(* PLC project PhysicsSimulator, Nammo OpenPLC 1 *)
(* stored: creationDateTime 2026-02-21T00:00:00, modificationDateTime 2026-02-21T00:00:00 *)

TYPE STATION_T : STRUCT
  number : INT;
  x_mm : REAL;
  station_type : INT;
  device_delay_s : REAL;
  dropping_time_s : REAL;
END_STRUCT;
END_TYPE

TYPE PHYSICS_2D_T : STRUCT
  x_accel_s : REAL;
  x_decel_s : REAL;
  x_max_mm_s : REAL;
  z_total_mm : REAL;
  z_slow_dry_mm : REAL;
  z_slow_wet_mm : REAL;
  z_slow_end_mm : REAL;
  z_slow_mm_s : REAL;
  z_fast_mm_s : REAL;
  drip_delay_s : REAL;
  avoid_mm : REAL;
END_STRUCT;
END_TYPE

TYPE TRANSPORTER_CFG_T : STRUCT
  id : INT;
  start_station : INT;
  x_min_limit : REAL;
  x_max_limit : REAL;
  phys2d : PHYSICS_2D_T;
END_STRUCT;
END_TYPE

TYPE TRANSPORTER_STATE_T : STRUCT
  active : BOOL;
  phase : INT;
  z_stage : INT;
  x_mm : REAL;
  z_mm : REAL;
  vel_x : REAL;
  vel_z : REAL;
  current_station : INT;
  lift_station_target : INT;
  sink_station_target : INT;
  target_x : REAL;
  x_min_limit : REAL;
  x_max_limit : REAL;
  z_timer_s : REAL;
END_STRUCT;
END_TYPE

FUNCTION IsWetStationType : BOOL
  VAR_INPUT
    station_type : INT;
  END_VAR

            IsWetStationType := (station_type = 1) OR (station_type = 11);
          
END_FUNCTION

FUNCTION_BLOCK FB_StationLookup
  VAR_INPUT
    station_number : INT;
  END_VAR
  VAR_OUTPUT
    found : BOOL;
    idx : INT;
    x_mm : REAL;
    stype : INT;
    device_delay_s : REAL;
    dropping_time_s : REAL;
  END_VAR
  VAR_EXTERNAL
    g_station_count : INT;
    g_stations : ARRAY[1..21] OF STATION_T;
  END_VAR
  VAR
    i : INT;
    tmp_st : STATION_T;
  END_VAR

            found := FALSE;
idx := 0;
x_mm := 0.0;
stype := 0;
device_delay_s := 0.0;
dropping_time_s := 0.0;

FOR i := 1 TO g_station_count DO
  tmp_st := g_stations[i];
  IF tmp_st.number = station_number THEN
    found := TRUE;
    idx := i;
    x_mm := tmp_st.x_mm;
    stype := tmp_st.station_type;
    device_delay_s := tmp_st.device_delay_s;
    dropping_time_s := tmp_st.dropping_time_s;
    RETURN;
  END_IF;
END_FOR;
          
END_FUNCTION_BLOCK

FUNCTION_BLOCK FB_XMotion
  VAR_INPUT
    delta_t : REAL;
    x_target : REAL;
    x_min : REAL;
    x_max : REAL;
    v_max : REAL;
    t_acc : REAL;
    t_dec : REAL;
  END_VAR
  VAR_IN_OUT
    x_pos : REAL;
    v_x : REAL;
  END_VAR
  VAR_OUTPUT
    arrived : BOOL;
  END_VAR
  VAR
    drive_target : REAL;
    distance : REAL;
    dir : REAL;
    a_acc : REAL;
    a_dec : REAL;
    brake_dist : REAL;
    new_vel : REAL;
    travel : REAL;
  END_VAR

            IF (x_max > x_min) THEN
  IF x_pos < x_min THEN
    drive_target := x_min;
  ELSIF x_pos > x_max THEN
    drive_target := x_max;
  ELSE
    IF x_target < x_min THEN
      drive_target := x_min;
    ELSIF x_target > x_max THEN
      drive_target := x_max;
    ELSE
      drive_target := x_target;
    END_IF;
  END_IF;
ELSE
  drive_target := x_target;
END_IF;

arrived := ABS(x_pos - drive_target) <= 3.0;
IF arrived THEN
  x_pos := drive_target;
  v_x := 0.0;
  RETURN;
END_IF;

IF t_acc <= 0.0 THEN t_acc := 0.001; END_IF;
IF t_dec <= 0.0 THEN t_dec := 0.001; END_IF;
IF v_max < 0.0 THEN v_max := 0.0; END_IF;

a_acc := v_max / t_acc;
a_dec := v_max / t_dec;

dir := 1.0;
IF drive_target < x_pos THEN
  dir := -1.0;
END_IF;

distance := ABS(drive_target - x_pos);

IF a_dec > 0.0 THEN
  brake_dist := (v_x * v_x) / (2.0 * a_dec);
ELSE
  brake_dist := 0.0;
END_IF;

IF brake_dist >= distance THEN
  new_vel := v_x - a_dec * delta_t;
  IF new_vel < 0.0 THEN new_vel := 0.0; END_IF;
ELSE
  new_vel := v_x + a_acc * delta_t;
  IF new_vel > v_max THEN new_vel := v_max; END_IF;
END_IF;

travel := new_vel * delta_t;
IF travel >= distance THEN
  x_pos := drive_target;
  v_x := 0.0;
  arrived := TRUE;
ELSE
  x_pos := x_pos + dir * travel;
  v_x := new_vel;
  arrived := FALSE;
END_IF;
          
END_FUNCTION_BLOCK

PROGRAM PLC_PRG
  VAR_EXTERNAL
    g_station_count : INT;
    g_stations : ARRAY[1..21] OF STATION_T;
    g_cfg : ARRAY[1..10] OF TRANSPORTER_CFG_T;
    g_state : ARRAY[1..10] OF TRANSPORTER_STATE_T;
    g_cmd_start : ARRAY[1..10] OF BOOL;
    g_cmd_lift_station : ARRAY[1..10] OF INT;
    g_cmd_sink_station : ARRAY[1..10] OF INT;
  END_VAR
  VAR
    init_done : BOOL := FALSE;
    i : INT;
    idx : INT;
    station_type : INT;
    device_delay : REAL;
    drop_time : REAL;
    slow_start : REAL;
    arrived_x : BOOL;
    nearest_num : INT;
    min_dist : REAL;
    dx : REAL;
    tmp_x : REAL;
    tmp_vx : REAL;
    fb_x1 : FB_XMotion;
    fb_x2 : FB_XMotion;
    lookup : FB_StationLookup;
  END_VAR

            IF NOT init_done THEN
  g_station_count := 21;

  g_stations[1].number := 101;
  g_stations[1].x_mm := 100.0;
  g_stations[1].station_type := 22;
  g_stations[1].device_delay_s := 0.0;
  g_stations[1].dropping_time_s := 0.0;

  g_stations[2].number := 102;
  g_stations[2].x_mm := 1550.0;
  g_stations[2].station_type := 30;
  g_stations[2].device_delay_s := 0.0;
  g_stations[2].dropping_time_s := 0.0;

  g_stations[3].number := 103;
  g_stations[3].x_mm := 3000.0;
  g_stations[3].station_type := 30;
  g_stations[3].device_delay_s := 0.0;
  g_stations[3].dropping_time_s := 0.0;

  g_stations[4].number := 104;
  g_stations[4].x_mm := 4450.0;
  g_stations[4].station_type := 0;
  g_stations[4].device_delay_s := 3.0;
  g_stations[4].dropping_time_s := 0.0;

  g_stations[5].number := 105;
  g_stations[5].x_mm := 5900.0;
  g_stations[5].station_type := 0;
  g_stations[5].device_delay_s := 3.0;
  g_stations[5].dropping_time_s := 0.0;

  g_stations[6].number := 106;
  g_stations[6].x_mm := 7350.0;
  g_stations[6].station_type := 0;
  g_stations[6].device_delay_s := 3.0;
  g_stations[6].dropping_time_s := 0.0;

  g_stations[7].number := 107;
  g_stations[7].x_mm := 8800.0;
  g_stations[7].station_type := 1;
  g_stations[7].device_delay_s := 3.0;
  g_stations[7].dropping_time_s := 10.0;

  g_stations[8].number := 108;
  g_stations[8].x_mm := 10250.0;
  g_stations[8].station_type := 1;
  g_stations[8].device_delay_s := 0.0;
  g_stations[8].dropping_time_s := 10.0;

  g_stations[9].number := 109;
  g_stations[9].x_mm := 11700.0;
  g_stations[9].station_type := 1;
  g_stations[9].device_delay_s := 0.0;
  g_stations[9].dropping_time_s := 10.0;

  g_stations[10].number := 110;
  g_stations[10].x_mm := 13150.0;
  g_stations[10].station_type := 1;
  g_stations[10].device_delay_s := 0.0;
  g_stations[10].dropping_time_s := 10.0;

  g_stations[11].number := 111;
  g_stations[11].x_mm := 14600.0;
  g_stations[11].station_type := 1;
  g_stations[11].device_delay_s := 0.0;
  g_stations[11].dropping_time_s := 10.0;

  g_stations[12].number := 112;
  g_stations[12].x_mm := 16050.0;
  g_stations[12].station_type := 1;
  g_stations[12].device_delay_s := 3.0;
  g_stations[12].dropping_time_s := 10.0;

  g_stations[13].number := 113;
  g_stations[13].x_mm := 17500.0;
  g_stations[13].station_type := 1;
  g_stations[13].device_delay_s := 0.0;
  g_stations[13].dropping_time_s := 10.0;

  g_stations[14].number := 114;
  g_stations[14].x_mm := 18950.0;
  g_stations[14].station_type := 32;
  g_stations[14].device_delay_s := 0.0;
  g_stations[14].dropping_time_s := 0.0;

  g_stations[15].number := 115;
  g_stations[15].x_mm := 20400.0;
  g_stations[15].station_type := 0;
  g_stations[15].device_delay_s := 3.0;
  g_stations[15].dropping_time_s := 10.0;

  g_stations[16].number := 116;
  g_stations[16].x_mm := 21850.0;
  g_stations[16].station_type := 1;
  g_stations[16].device_delay_s := 3.0;
  g_stations[16].dropping_time_s := 10.0;

  g_stations[17].number := 117;
  g_stations[17].x_mm := 23300.0;
  g_stations[17].station_type := 1;
  g_stations[17].device_delay_s := 0.0;
  g_stations[17].dropping_time_s := 10.0;

  g_stations[18].number := 118;
  g_stations[18].x_mm := 24750.0;
  g_stations[18].station_type := 1;
  g_stations[18].device_delay_s := 0.0;
  g_stations[18].dropping_time_s := 10.0;

  g_stations[19].number := 119;
  g_stations[19].x_mm := 26200.0;
  g_stations[19].station_type := 30;
  g_stations[19].device_delay_s := 0.0;
  g_stations[19].dropping_time_s := 0.0;

  g_stations[20].number := 120;
  g_stations[20].x_mm := 27650.0;
  g_stations[20].station_type := 30;
  g_stations[20].device_delay_s := 0.0;
  g_stations[20].dropping_time_s := 0.0;

  g_stations[21].number := 121;
  g_stations[21].x_mm := 29100.0;
  g_stations[21].station_type := 1;
  g_stations[21].device_delay_s := 0.0;
  g_stations[21].dropping_time_s := 10.0;

  g_cfg[1].id := 1;
  g_cfg[1].start_station := 101;
  g_cfg[1].x_min_limit := 100.0;
  g_cfg[1].x_max_limit := 20600.0;
  g_cfg[1].phys2d.x_accel_s := 1.5;
  g_cfg[1].phys2d.x_decel_s := 1.5;
  g_cfg[1].phys2d.x_max_mm_s := 500.0;
  g_cfg[1].phys2d.z_total_mm := 2500.0;
  g_cfg[1].phys2d.z_slow_dry_mm := 300.0;
  g_cfg[1].phys2d.z_slow_wet_mm := 1000.0;
  g_cfg[1].phys2d.z_slow_end_mm := 50.0;
  g_cfg[1].phys2d.z_slow_mm_s := 100.0;
  g_cfg[1].phys2d.z_fast_mm_s := 200.0;
  g_cfg[1].phys2d.drip_delay_s := 5.0;
  g_cfg[1].phys2d.avoid_mm := 2000.0;

  g_cfg[2].id := 2;
  g_cfg[2].start_station := 118;
  g_cfg[2].x_min_limit := 14300.0;
  g_cfg[2].x_max_limit := 29100.0;
  g_cfg[2].phys2d.x_accel_s := 1.5;
  g_cfg[2].phys2d.x_decel_s := 1.5;
  g_cfg[2].phys2d.x_max_mm_s := 500.0;
  g_cfg[2].phys2d.z_total_mm := 2500.0;
  g_cfg[2].phys2d.z_slow_dry_mm := 300.0;
  g_cfg[2].phys2d.z_slow_wet_mm := 1000.0;
  g_cfg[2].phys2d.z_slow_end_mm := 50.0;
  g_cfg[2].phys2d.z_slow_mm_s := 100.0;
  g_cfg[2].phys2d.z_fast_mm_s := 200.0;
  g_cfg[2].phys2d.drip_delay_s := 5.0;
  g_cfg[2].phys2d.avoid_mm := 2000.0;

  FOR i := 1 TO 10 DO
    IF i <= 2 THEN
      g_state[i].active := TRUE;
    ELSE
      g_state[i].active := FALSE;
    END_IF;
    g_state[i].phase := 0;
    g_state[i].z_stage := 0;
    g_state[i].vel_x := 0.0;
    g_state[i].vel_z := 0.0;
    g_state[i].z_timer_s := 0.0;
    g_state[i].x_min_limit := g_cfg[i].x_min_limit;
    g_state[i].x_max_limit := g_cfg[i].x_max_limit;

    lookup(station_number := g_cfg[i].start_station);
    IF lookup.found THEN
      g_state[i].x_mm := lookup.x_mm;
      g_state[i].current_station := g_cfg[i].start_station;
    ELSE
      g_state[i].x_mm := 0.0;
      g_state[i].current_station := 0;
    END_IF;
    g_state[i].z_mm := 0.0;
  END_FOR;

  init_done := TRUE;
END_IF;

FOR i := 1 TO 10 DO
  IF g_state[i].active THEN

  IF (g_state[i].phase = 0) AND g_cmd_start[i] THEN
    g_state[i].lift_station_target := g_cmd_lift_station[i];
    g_state[i].sink_station_target := g_cmd_sink_station[i];
    lookup(station_number := g_state[i].lift_station_target);
    g_state[i].target_x := lookup.x_mm;
    g_state[i].phase := 1;
    g_state[i].z_stage := 0;
    g_state[i].z_timer_s := 0.0;
  END_IF;

  IF g_state[i].phase = 1 THEN
    tmp_x := g_state[i].x_mm;
    tmp_vx := g_state[i].vel_x;
    IF i = 1 THEN
      fb_x1(
        delta_t := 0.02,
        x_target := g_state[i].target_x,
        x_min := g_state[i].x_min_limit,
        x_max := g_state[i].x_max_limit,
        v_max := g_cfg[i].phys2d.x_max_mm_s,
        t_acc := g_cfg[i].phys2d.x_accel_s,
        t_dec := g_cfg[i].phys2d.x_decel_s,
        x_pos := tmp_x,
        v_x := tmp_vx
      );
      arrived_x := fb_x1.arrived;
    ELSIF i = 2 THEN
      fb_x2(
        delta_t := 0.02,
        x_target := g_state[i].target_x,
        x_min := g_state[i].x_min_limit,
        x_max := g_state[i].x_max_limit,
        v_max := g_cfg[i].phys2d.x_max_mm_s,
        t_acc := g_cfg[i].phys2d.x_accel_s,
        t_dec := g_cfg[i].phys2d.x_decel_s,
        x_pos := tmp_x,
        v_x := tmp_vx
      );
      arrived_x := fb_x2.arrived;
    END_IF;
    g_state[i].x_mm := tmp_x;
    g_state[i].vel_x := tmp_vx;

    IF arrived_x THEN
      g_state[i].current_station := g_state[i].lift_station_target;
      lookup(station_number := g_state[i].lift_station_target);
      device_delay := lookup.device_delay_s;
      drop_time := lookup.dropping_time_s;
      g_state[i].z_timer_s := device_delay + drop_time;
      g_state[i].z_stage := 1;
      g_state[i].phase := 2;
    END_IF;
  END_IF;

  IF g_state[i].phase = 2 THEN
    lookup(station_number := g_state[i].lift_station_target);
    station_type := lookup.stype;
    IF IsWetStationType(station_type) THEN
      slow_start := g_cfg[i].phys2d.z_slow_wet_mm;
    ELSE
      slow_start := g_cfg[i].phys2d.z_slow_dry_mm;
    END_IF;

    CASE g_state[i].z_stage OF
      1:
        g_state[i].z_timer_s := g_state[i].z_timer_s - 0.02;
        IF g_state[i].z_timer_s <= 0.0 THEN
          g_state[i].z_stage := 2;
          g_state[i].z_mm := g_cfg[i].phys2d.z_total_mm;
        END_IF;
      2:
        g_state[i].z_mm := g_state[i].z_mm - g_cfg[i].phys2d.z_slow_mm_s * 0.02;
        IF g_state[i].z_mm <= (g_cfg[i].phys2d.z_total_mm - slow_start) THEN
          g_state[i].z_stage := 3;
        END_IF;
      3:
        g_state[i].z_mm := g_state[i].z_mm - g_cfg[i].phys2d.z_fast_mm_s * 0.02;
        IF g_state[i].z_mm <= g_cfg[i].phys2d.z_slow_end_mm THEN
          g_state[i].z_stage := 4;
        END_IF;
      4:
        g_state[i].z_mm := g_state[i].z_mm - g_cfg[i].phys2d.z_slow_mm_s * 0.02;
        IF g_state[i].z_mm <= 0.0 THEN
          g_state[i].z_mm := 0.0;
          g_state[i].z_timer_s := g_cfg[i].phys2d.drip_delay_s;
          g_state[i].z_stage := 5;
        END_IF;
      5:
        g_state[i].z_timer_s := g_state[i].z_timer_s - 0.02;
        IF g_state[i].z_timer_s <= 0.0 THEN
          g_state[i].z_stage := 0;
          lookup(station_number := g_state[i].sink_station_target);
          g_state[i].target_x := lookup.x_mm;
          g_state[i].phase := 3;
        END_IF;
    END_CASE;
  END_IF;

  IF g_state[i].phase = 3 THEN
    tmp_x := g_state[i].x_mm;
    tmp_vx := g_state[i].vel_x;
    IF i = 1 THEN
      fb_x1(
        delta_t := 0.02,
        x_target := g_state[i].target_x,
        x_min := g_state[i].x_min_limit,
        x_max := g_state[i].x_max_limit,
        v_max := g_cfg[i].phys2d.x_max_mm_s,
        t_acc := g_cfg[i].phys2d.x_accel_s,
        t_dec := g_cfg[i].phys2d.x_decel_s,
        x_pos := tmp_x,
        v_x := tmp_vx
      );
      arrived_x := fb_x1.arrived;
    ELSIF i = 2 THEN
      fb_x2(
        delta_t := 0.02,
        x_target := g_state[i].target_x,
        x_min := g_state[i].x_min_limit,
        x_max := g_state[i].x_max_limit,
        v_max := g_cfg[i].phys2d.x_max_mm_s,
        t_acc := g_cfg[i].phys2d.x_accel_s,
        t_dec := g_cfg[i].phys2d.x_decel_s,
        x_pos := tmp_x,
        v_x := tmp_vx
      );
      arrived_x := fb_x2.arrived;
    END_IF;
    g_state[i].x_mm := tmp_x;
    g_state[i].vel_x := tmp_vx;

    IF arrived_x THEN
      g_state[i].current_station := g_state[i].sink_station_target;
      lookup(station_number := g_state[i].sink_station_target);
      device_delay := lookup.device_delay_s;
      g_state[i].z_timer_s := device_delay + g_cfg[i].phys2d.drip_delay_s;
      g_state[i].z_stage := 6;
      g_state[i].phase := 4;
    END_IF;
  END_IF;

  IF g_state[i].phase = 4 THEN
    lookup(station_number := g_state[i].sink_station_target);
    station_type := lookup.stype;
    IF IsWetStationType(station_type) THEN
      slow_start := g_cfg[i].phys2d.z_slow_wet_mm;
    ELSE
      slow_start := g_cfg[i].phys2d.z_slow_dry_mm;
    END_IF;

    CASE g_state[i].z_stage OF
      6:
        g_state[i].z_timer_s := g_state[i].z_timer_s - 0.02;
        IF g_state[i].z_timer_s <= 0.0 THEN
          g_state[i].z_stage := 7;
        END_IF;
      7:
        g_state[i].z_mm := g_state[i].z_mm + g_cfg[i].phys2d.z_fast_mm_s * 0.02;
        IF g_state[i].z_mm >= (g_cfg[i].phys2d.z_total_mm - slow_start) THEN
          g_state[i].z_stage := 8;
        END_IF;
      8:
        g_state[i].z_mm := g_state[i].z_mm + g_cfg[i].phys2d.z_slow_mm_s * 0.02;
        IF g_state[i].z_mm >= g_cfg[i].phys2d.z_total_mm THEN
          g_state[i].z_mm := g_cfg[i].phys2d.z_total_mm;
          g_state[i].z_stage := 0;
          g_state[i].phase := 0;
        END_IF;
    END_CASE;
  END_IF;

  min_dist := 1.0e9;
  nearest_num := g_state[i].current_station;
  FOR idx := 1 TO g_station_count DO
    dx := g_stations[idx].x_mm - g_state[i].x_mm;
    IF ABS(dx) < min_dist THEN
      min_dist := ABS(dx);
      nearest_num := g_stations[idx].number;
    END_IF;
  END_FOR;
  g_state[i].current_station := nearest_num;

  END_IF;
END_FOR;
          
END_PROGRAM

CONFIGURATION Config0
  VAR_GLOBAL
    g_station_count : INT := 0;
    g_stations : ARRAY[1..21] OF STATION_T;
    g_cfg : ARRAY[1..10] OF TRANSPORTER_CFG_T;
    g_state : ARRAY[1..10] OF TRANSPORTER_STATE_T;
    g_cmd_start : ARRAY[1..10] OF BOOL;
    g_cmd_lift_station : ARRAY[1..10] OF INT;
    g_cmd_sink_station : ARRAY[1..10] OF INT;
  END_VAR
  RESOURCE Res0 ON PLC
    TASK task0(INTERVAL := T#20ms, PRIORITY := 0);
    PROGRAM instance0 WITH task0 : PLC_PRG;
  END_RESOURCE
END_CONFIGURATION
